{attribute 'no_assign'}
{attribute 'enable_dynamic_creation'}
{attribute 'no_explicit_call' := 'do not call this POU directly'}
{attribute 'reflection'} 
FUNCTION_BLOCK CStringBuilder IMPLEMENTS I_StringBuilder
VAR_INPUT
END_VAR
VAR_OUTPUT
END_VAR
VAR
	pBuffer : POINTER TO BYTE;
	_maxBufferSize : UDINT; //defines max possible string length
	_currentUsedBufferSize : UDINT;
	
	{attribute 'instance-path'} 
    {attribute 'noinit'} 
    sPath : STRING; 
END_VAR

METHOD AnyToString : STRING
VAR_INPUT
	Value : ANY;
END_VAR
VAR
	pBool			: POINTER TO BOOL;
    pByte			: POINTER TO BYTE;
    pWord			: POINTER TO WORD;
    pDWord			: POINTER TO DWORD;
    pLWord			: POINTER TO LWORD;
    pSint			: POINTER TO SINT;
    pInt			: POINTER TO INT;
    pDint			: POINTER TO DINT;
    pLint			: POINTER TO LINT;
    pUSint			: POINTER TO USINT;
    pUInt			: POINTER TO UINT;
    pUDint			: POINTER TO UDINT;
    pULint			: POINTER TO ULINT;
    pReal			: POINTER TO REAL;
    pLReal			: POINTER TO LREAL;
    pString			: POINTER TO T_MaxString;
    pWString		: POINTER TO WSTRING;
    pTime			: POINTER TO TIME;
    pDate			: POINTER TO DATE;
    pDateAndTime	: POINTER TO DATE_AND_TIME;
    pTimeOfDay		: POINTER TO TIME_OF_DAY;
    pPointer		: PVOID;
	pLTime 			: POINTER TO LTIME;
END_VAR
IF Value.pValue = 0 THEN RETURN; END_IF;

CASE Value.TypeClass OF 
	__SYSTEM.TYPE_CLASS.TYPE_BOOL:
		pBool := Value.pValue;
		AnyToString := TO_STRING(pBool^);
		
    __SYSTEM.TYPE_CLASS.TYPE_BYTE:
		pByte := Value.pValue;
		AnyToString := TO_STRING(pByte^);
		
    __SYSTEM.TYPE_CLASS.TYPE_WORD:
		pWord := Value.pValue;
		AnyToString := TO_STRING(pWord^);
		
    __SYSTEM.TYPE_CLASS.TYPE_DWORD:
		pDWord := Value.pValue;
		AnyToString := TO_STRING(pDWord^);
		
    __SYSTEM.TYPE_CLASS.TYPE_LWORD:
		pLWord := Value.pValue;
		AnyToString := TO_STRING(pLWord^);
		
    __SYSTEM.TYPE_CLASS.TYPE_SINT:
		pSint := Value.pValue;
		AnyToString := TO_STRING(pSint^);
		
    __SYSTEM.TYPE_CLASS.TYPE_INT:
		pInt := Value.pValue;
		AnyToString := TO_STRING(pInt^);
		
    __SYSTEM.TYPE_CLASS.TYPE_DINT:
		pDint := Value.pValue;
		AnyToString := TO_STRING(pDint^);
		
    __SYSTEM.TYPE_CLASS.TYPE_LINT:
		pLint := Value.pValue;
		AnyToString := TO_STRING(pLint^);
		
    __SYSTEM.TYPE_CLASS.TYPE_USINT:
		pUSint := Value.pValue;
		AnyToString := TO_STRING(pUSint^);
		
    __SYSTEM.TYPE_CLASS.TYPE_UINT:
		pUInt := Value.pValue;
		AnyToString := TO_STRING(pUInt^);
		
    __SYSTEM.TYPE_CLASS.TYPE_UDINT:
		pUDint := Value.pValue;
		AnyToString := TO_STRING(pUDint^);
		
    __SYSTEM.TYPE_CLASS.TYPE_ULINT:
		pULint := Value.pValue;
		AnyToString := TO_STRING(pULint^);
		
   __SYSTEM.TYPE_CLASS.TYPE_REAL:
		pReal := Value.pValue;
		AnyToString := TO_STRING(pReal^);
		
    __SYSTEM.TYPE_CLASS.TYPE_LREAL:
		pLReal := Value.pValue;
		AnyToString := TO_STRING(pLReal^);
		
    __SYSTEM.TYPE_CLASS.TYPE_STRING:
		pString := Value.pValue;
		AnyToString := TO_STRING(pString^);
		
   __SYSTEM.TYPE_CLASS.TYPE_WSTRING:
		pWString := Value.pValue;
		AnyToString := TO_STRING(pWString^);
		
    __SYSTEM.TYPE_CLASS.TYPE_TIME:
		pTime := Value.pValue;
		AnyToString := TO_STRING(pTime^);
		
    __SYSTEM.TYPE_CLASS.TYPE_DATE:
		pDate := Value.pValue;
		AnyToString := TO_STRING(pDate^);
		
    __SYSTEM.TYPE_CLASS.TYPE_DATEANDTIME:
		pDateAndTime := Value.pValue;
		AnyToString := TO_STRING(pDateAndTime^);
		
    __SYSTEM.TYPE_CLASS.TYPE_TIMEOFDAY:
		pTimeOfDay := Value.pValue;
		AnyToString := TO_STRING(pTimeOfDay^);
	
	__SYSTEM.TYPE_CLASS.TYPE_POINTER:
		AnyToString := TO_STRING(Value.pValue);
		
	__SYSTEM.TYPE_CLASS.TYPE_LTIME:
		pLTime := Value.pValue;
		AnyToString := TO_STRING(pLTime^);
ELSE
	RETURN; 
END_CASE
END_METHOD

METHOD Append : I_StringBuilder
VAR_INPUT
	Value : T_MaxString;
END_VAR
Append := THIS^.AppendAny(Value);
END_METHOD

// Appends the given value to the end of the string builder's contents.
METHOD AppendAny : I_StringBuilder
VAR_INPUT
	Value : ANY;
END_VAR
VAR
	stringLength : UDINT;
	convertedAny : STRING; 
	pValue : POINTER TO BYTE;
END_VAR
AppendAny := THIS^;

IF THIS^.pBuffer = 0 THEN
	ADSLOGSTR(msgCtrlMask:= ADSLOG_MSGTYPE_ERROR, msgFmtStr:='Dynamic buffer null pointer, usage of StringBuilder not possible', '');
	RETURN;
END_IF

CASE Value.TypeClass OF
	__SYSTEM.TYPE_CLASS.TYPE_STRING: 
		pValue := Value.pValue;
		
	__SYSTEM.TYPE_CLASS.TYPE_BOOL,
	__SYSTEM.TYPE_CLASS.TYPE_BYTE,
	__SYSTEM.TYPE_CLASS.TYPE_WORD,
	__SYSTEM.TYPE_CLASS.TYPE_DWORD,
	__SYSTEM.TYPE_CLASS.TYPE_LWORD,
	__SYSTEM.TYPE_CLASS.TYPE_SINT,
	__SYSTEM.TYPE_CLASS.TYPE_INT,
	__SYSTEM.TYPE_CLASS.TYPE_DINT,
	__SYSTEM.TYPE_CLASS.TYPE_LINT,
	__SYSTEM.TYPE_CLASS.TYPE_USINT,
	__SYSTEM.TYPE_CLASS.TYPE_UINT,
	__SYSTEM.TYPE_CLASS.TYPE_UDINT,
	__SYSTEM.TYPE_CLASS.TYPE_ULINT,
	__SYSTEM.TYPE_CLASS.TYPE_REAL,
	__SYSTEM.TYPE_CLASS.TYPE_LREAL,
	__SYSTEM.TYPE_CLASS.TYPE_TIME,
	__SYSTEM.TYPE_CLASS.TYPE_LTIME,
	__SYSTEM.TYPE_CLASS.TYPE_DATE,
	__SYSTEM.TYPE_CLASS.TYPE_DATEANDTIME,
	__SYSTEM.TYPE_CLASS.TYPE_TIMEOFDAY,
	__SYSTEM.TYPE_CLASS.TYPE_POINTER:
		convertedAny := AnyToString(Value);
		pValue := ADR(convertedAny);
ELSE
	RETURN;
END_CASE

stringLength := GetUsedStringLength(pByte:=pValue);

//check available size, existing size
IF stringLength = 0 THEN
	RETURN;
END_IF
//only copy if we do not exceed possible limit
IF THIS^._currentUsedBufferSize + stringLength >= THIS^._maxBufferSize THEN
	RETURN;
END_IF
MEMCPY(destAddr:=(THIS^.pBuffer + THIS^._currentUsedBufferSize), srcAddr:=pValue, n:=stringLength);

THIS^._currentUsedBufferSize := THIS^._currentUsedBufferSize + stringLength;
END_METHOD

PROPERTY BufferAddress : POINTER TO BYTE
GET
BufferAddress := THIS^.pBuffer;
END_GET
END_PROPERTY

METHOD Clear : I_StringBuilder
VAR_INPUT
END_VAR
Clear := THIS^;
IF THIS^.pBuffer = 0 THEN
	RETURN;
END_IF

MEMSET(destAddr:=THIS^.pBuffer, fillByte:=0, n:=THIS^.MaxBufferSize);
END_METHOD

PROPERTY CurrentBufferSize : UDINT
GET
CurrentBufferSize := THIS^._currentUsedBufferSize;
END_GET
END_PROPERTY

METHOD GetUsedStringLength : UDINT
VAR_INPUT
	pByte : POINTER TO BYTE;
END_VAR
VAR
    i : UDINT := 0;
END_VAR
//every string in twincat is 0 terminated
IF pByte = 0 THEN
	RETURN;
END_IF

WHILE (pByte^ <> 0) DO
    pByte := pByte + 1; // Pointer auf das nächste Byte verschieben
    i := i + 1;
END_WHILE;

GetUsedStringLength := i;
END_METHOD

METHOD Init : I_StringBuilder
VAR_INPUT
	pPara : POINTER TO ST_StringBuilderPara;
END_VAR
// TODO: add logging for failed allocation
IF ParaErrors(pPara:=pPara) THEN
	RETURN;
END_IF

IF THIS^.pBuffer <> 0 THEN
	__DELETE(THIS^.pBuffer);
END_IF

THIS^.pBuffer := __NEW(BYTE, pPara^.MaxBufferSize);
THIS^._maxBufferSize := pPara^.MaxBufferSize;
END_METHOD

PROPERTY MaxBufferSize : UDINT
GET
MaxBufferSize := THIS^._maxBufferSize;
END_GET
END_PROPERTY

{attribute 'reflection'} 
METHOD PRIVATE ParaErrors : BOOL
VAR_INPUT
	pPara : POINTER TO ST_StringBuilderPara;
END_VAR
VAR
	s1 : STRING(35) := 'Invalid parametrization pointer at ';
	s2: T_MaxString;
END_VAR
IF pPara = 0 THEN
	CONCAT2(pSrcString1:=ADR(s1), pSrcString2:=ADR(THIS^.sPath), pDstString:=ADR(s2), nDstSize:=SIZEOF(s2));
	ADSLOGSTR(msgCtrlMask:= ADSLOG_MSGTYPE_ERROR, msgFmtStr:=s2, '');
	ParaErrors := TRUE;
	RETURN;
END_IF
IF pPara^.MaxBufferSize = 0 THEN
	s1 := 'BufferSize 0 given, Stringbuilder init failed at ';
	CONCAT2(pSrcString1:=ADR(s1), pSrcString2:=ADR(THIS^.sPath), pDstString:=ADR(s2), nDstSize:=SIZEOF(s2));
	ADSLOGSTR(msgCtrlMask:= ADSLOG_MSGTYPE_ERROR, msgFmtStr:=s2, '');
	ParaErrors := TRUE;
	RETURN;
END_IF
END_METHOD

METHOD Reset : I_StringBuilder
VAR_INPUT
	pPara : POINTER TO ST_StringBuilderPara;
END_VAR
Reset := THIS^;
Clear();

IF ParaErrors(pPara:=pPara) THEN
	RETURN;
END_IF

Init(pPara:=pPara);
END_METHOD

END_FUNCTION_BLOCK

(* stored: Version 1.1.0.1, ProductVersion 3.1.4024.13
   POU CStringBuilder: Id {79373a45-1f4b-49ff-bd8a-456d74f0dd44}, SpecialFunc None
   Method AnyToString: Id {5ead9a6d-2f38-4e44-8a90-6d0ccb4b52ed}
   Method Append: Id {474915fc-a233-4555-a235-ca409caaa38d}
   Method AppendAny: Id {bd1b6489-49b2-0096-26d8-3075aa66e4a8}
   Property BufferAddress: Id {a5fb5549-c08a-4c47-8603-5eb042025092}
   Get Get: Id {07c0f9ec-d4a4-48d3-adbc-6862f32f272f}
   Method Clear: Id {027044e4-4377-4c44-9597-421e0eeb6261}
   Property CurrentBufferSize: Id {81e32561-fd56-4c8d-a3f6-4b792bb65c46}
   Get Get: Id {fd79a365-f513-441f-9fae-cf28cdbe0b18}
   Method GetUsedStringLength: Id {d2916a93-b823-422f-aa12-59c615f2b767}
   Method Init: Id {a6ff0c47-f3ea-4483-8981-c259eb39a22c}
   Property MaxBufferSize: Id {cd6561ae-aca3-438b-a685-cbb63239aa56}
   Get Get: Id {0d67c07e-bac9-47d4-9ccb-9b715c3a7fe9}
   Method ParaErrors: Id {17c190cc-4470-4fb6-af3d-cbed72e8f47a}
   Method Reset: Id {89de333b-4dc5-4a97-80a0-6f8c11f6e476} *)
